// TIA Portal project "time_delay_interrupt" (V18)

(* hardware
DEVICE "S7-1200 station_1"  S7-1200 Station
   slot 0: "Rack_0"  S7-1200 Rack  Rack  V1.0
   slot 1: "PLC_1"  CPU 1214C DC/DC/DC  6ES7 214-1AG40-0XB0  V4.6
*)

// ===== PLC "PLC_1"  CPU 1214C DC/DC/DC =====

VAR_GLOBAL   // PLC tag table "Default tag table"
   "Tag_1" AT %I0.0 : Bool;
   "Tag_2" AT %M10.0 : Bool;
   "Tag_3" AT %MW20 : Word;
   "Tag_4" AT %MW0 : Int;
   "Tag_5" AT %I0.1 : Bool;
   "Tag_6" AT %MW4 : Int;
   "Tag_7" AT %MW6 : Int;
   "Tag_8" AT %MW8 : Word;
END_VAR

ORGANIZATION_BLOCK "Main"   // OB1, LAD, ProgramCycle
TITLE = "Main Program Sweep (Cycle)"
{ S7_Optimized_Access := 'TRUE' }
VERSION : 0.1
   VAR_INPUT
      Initial_Call : Bool;   // Initial call of this OB
      Remanence : Bool;   // =True, if remanent data are available
   END_VAR
BEGIN
END_ORGANIZATION_BLOCK

ORGANIZATION_BLOCK "Time delay interrupt"   // OB20, LAD, TimeDelayInterrupt
{ S7_Optimized_Access := 'TRUE' }
VERSION : 0.1
// extended instrution menüsünden al
// 
// srt_dint ile kesme işlemi başlatılır
// an_dint ile kesme işlemi durdurulur
// qry_dint ile kesme durumu sorgulanır
   VAR_INPUT
      Sign : Word;   // Identifier input (SIGN) passed to triggering call of SRT_DINT
   END_VAR
   VAR_TEMP   // added for the SCL form of the ladder/FBD networks
      _w1 : Bool;
   END_VAR
BEGIN

REGION Network 1
   // ob_nr numara
   // dtime süre sonunda bir kez kesme çalışır
   // sign ın s71200 için bir anlamı yoktur
   // ret_wall 0000 ise ata yoktur- 80 -90 görmüşsek hata geçersizdir
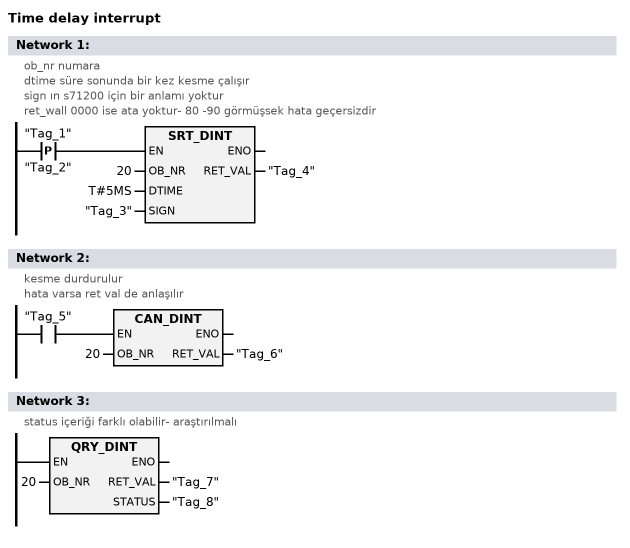
   #_w1 := "Tag_1" AND NOT "Tag_2";   // rising edge of "Tag_1"
   "Tag_2" := "Tag_1";
   IF #_w1 THEN "Tag_4" := SRT_DINT(OB_NR := 20, DTIME := T#5MS, SIGN := "Tag_3"); END_IF;
END_REGION

REGION Network 2
   // kesme durdurulur
   // hata varsa ret val de anlaşılır
   IF "Tag_5" THEN "Tag_6" := CAN_DINT(OB_NR := 20); END_IF;
END_REGION

REGION Network 3
   // status içeriği farklı olabilir- araştırılmalı
   "Tag_7" := QRY_DINT(OB_NR := 20, STATUS => "Tag_8");
END_REGION
END_ORGANIZATION_BLOCK